Yaskawa INFORM job: STKCOPY.JBI

/JOB
//NAME STKCOPY
///FOLDERNAME SpeedbotUnStack
//POS
///NPOS 0,0,0,10,0,0
///TOOL 0
///POSTYPE BASE
///RECTAN
///RCONF 1,0,0,0,0,0,0,0,0,0,0,0,0,0,0,0,0,0,0,0,0,0,0,0
P00031=793.061,-0.005,327.918,179.9626,7.7053,-0.0048
P00032=793.061,-0.005,327.918,179.9626,7.7053,-0.0048
///RCONF 0,0,0,0,0,0,0,0,0,0,0,0,0,0,0,0,0,0,0,0,0,0,0,0
P00050=0.000,0.000,0.000,0.0000,0.0000,0.0000
P00051=0.000,0.000,0.000,0.0000,0.0000,0.0000
P00052=0.000,0.000,0.000,0.0000,0.0000,0.0000
P00056=0.000,0.000,0.000,0.0000,0.0000,0.0000
P00057=0.000,0.000,0.000,0.0000,0.0000,0.0000
P00060=0.000,0.000,0.000,0.0000,0.0000,0.0000
P00061=0.000,0.000,0.000,0.0000,0.0000,0.0000
P00062=0.000,0.000,0.000,0.0000,0.0000,0.0000
//INST
///DATE 2025/04/20 22:24
///ATTR SC,RW
///GROUP1 RB1
///LVARS 10,10,10,10,10,10,0,0
NOP
'Part Id
SET D050 D060
'Area Id
SET D051 D061
'Grip Pip
SET D052 D062
'Heigth
SET R050 R060
'Windth
SET R051 R061
'Hig
SET R052 R062
'Pick Pos
SET P050 P060
'Place Pos
SET P051 P061
'Obli Pos
SET P052 P062
'抓取接近点
MULMAT P056 P050 P031
'抓取离开点
MULMAT P057 P050 P032
END
